// minimal transport for the connector base suite
FUNCTION_BLOCK FB_ProbeConnector EXTENDS FB_DeviceConnectorBase
VAR_INPUT
    SimOpenOk : BOOL := TRUE;
    SimHb     : E_HbResult := E_HbResult.OK;
END_VAR

Cyclic();

METHOD PROTECTED _M_Close : BOOL
_M_Close := TRUE;
END_METHOD

METHOD PROTECTED _M_HbPoll : E_HbResult
_M_HbPoll := SimHb;
END_METHOD

METHOD PROTECTED _M_HbStart : BOOL
_M_HbStart := TRUE;
END_METHOD

METHOD PROTECTED _M_Open : BOOL
_M_Open := SimOpenOk;
END_METHOD

END_FUNCTION_BLOCK

(* stored: Version 1.1.0.1, ProductVersion 3.1.4024.12
   POU FB_ProbeConnector: Id {c59dfe4e-41d8-46f2-8e29-cd61ea27b721}, SpecialFunc None
   Method _M_Close: Id {fa6aa4d5-061c-42cf-a901-aca4f5dc4c47}
   Method _M_HbPoll: Id {dbda08f4-7a78-44ab-8f25-81876beaeda9}
   Method _M_HbStart: Id {324ff04c-82eb-40aa-88f8-d148cf35637c}
   Method _M_Open: Id {508ced4c-bc17-44b5-8420-96a7b685819f} *)
